_CFC_ (* Continuous Function Chart, elements in execution order *)
(* 50с *)
#0 INT_TO_TIME(SCHU_P2_3_YA2_ZADER_RAS_DOST)
#1 MUL(#0, 1000)
#2 TON_YA2_Rassog1:TON(IN: YA2_DOST, PT: #1)
#3 ABS(SCHU_P2_3_YA2_RASSOG)
#4 GT(#3, SCHU_P2_3_YA2_UST_RASSOG)
#5 GT(SCHU_P2_3_YA2_RASSOG, SCHU_P2_3_YA2_UST_RASSOG)
#6 SEL(SCHU_P2_3_UST_RE_STOP, #4, #5)
#7 ABS(SCHU_P2_3_YA2_RASSOG_POL)
#8 GT(#7, SCHU_P2_3_YA2_UST_RASSOG)
#9 AND(TRUE, #8)
#10 YA2_REG_POL <= #9
#11 SEL(YA2_REG_POL, #6, #8)
#12 AND(NOT SCHU_P2_3_UST_RE_PUSK, #11)
#13 INT_TO_TIME(SCHU_P2_3_YA2_ZADER_RAS)
#14 MUL(#13, 1000)
#15 TON_YA2_Rassog:TON(IN: #12, PT: #14)
#16 OR(#15.Q, YA2_AO_OTKAZ)
#17 AND(#2.Q, SCHU_P2_3_SA4_DI3_A, #16)
#18 SR_YA2_Otk:SR(SET1: #17, RESET: SCHU_P2_3_SB)
#19 SCHU_P2_3_Z_YA2_OTKAZ <= #18.Q1
_END_CFC_
(* the same logic as Structured Text *)
(* 50с *)
TON_YA2_Rassog1(IN := YA2_DOST, PT := INT_TO_TIME(SCHU_P2_3_YA2_ZADER_RAS_DOST) * 1000);
_t14 := ABS(SCHU_P2_3_YA2_RASSOG_POL) > SCHU_P2_3_YA2_UST_RASSOG;
YA2_REG_POL := TRUE AND _t14;
TON_YA2_Rassog(IN := NOT SCHU_P2_3_UST_RE_PUSK AND SEL(YA2_REG_POL, SEL(SCHU_P2_3_UST_RE_STOP, ABS(SCHU_P2_3_YA2_RASSOG) > SCHU_P2_3_YA2_UST_RASSOG, SCHU_P2_3_YA2_RASSOG > SCHU_P2_3_YA2_UST_RASSOG), _t14), PT := INT_TO_TIME(SCHU_P2_3_YA2_ZADER_RAS) * 1000);
SR_YA2_Otk(SET1 := TON_YA2_Rassog1.Q AND SCHU_P2_3_SA4_DI3_A AND (TON_YA2_Rassog.Q OR YA2_AO_OTKAZ), RESET := SCHU_P2_3_SB);
SCHU_P2_3_Z_YA2_OTKAZ := SR_YA2_Otk.Q1;
END_PROGRAM

(* POU TZBiS/TZB/Z_YA3_Otk, CFC *)
PROGRAM Z_YA3_Otk
VAR
	SR_YA3_Otk: SR;
	TON_YA3_Zakl: TON;
	TON_YA3_Rassog: TON;
END_VAR
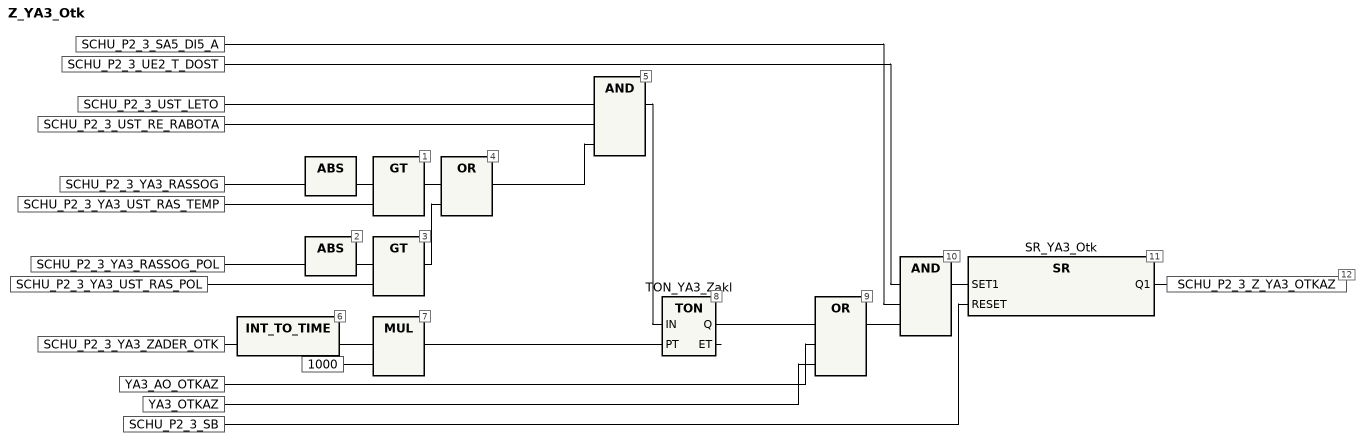
_CFC_ (* Continuous Function Chart, elements in execution order *)
#0 ABS(SCHU_P2_3_YA3_RASSOG)
#1 GT(#0, SCHU_P2_3_YA3_UST_RAS_TEMP)
#2 ABS(SCHU_P2_3_YA3_RASSOG_POL)
#3 GT(#2, SCHU_P2_3_YA3_UST_RAS_POL)
#4 OR(#1, #3)
#5 AND(SCHU_P2_3_UST_LETO, SCHU_P2_3_UST_RE_RABOTA, #4)
#6 INT_TO_TIME(SCHU_P2_3_YA3_ZADER_OTK)
#7 MUL(#6, 1000)
#8 TON_YA3_Zakl:TON(IN: #5, PT: #7)
#9 OR(#8.Q, YA3_AO_OTKAZ, YA3_OTKAZ)
#10 AND(SCHU_P2_3_UE2_T_DOST, SCHU_P2_3_SA5_DI5_A, #9)
#11 SR_YA3_Otk:SR(SET1: #10, RESET: SCHU_P2_3_SB)
#12 SCHU_P2_3_Z_YA3_OTKAZ <= #11.Q1
_END_CFC_
(* the same logic as Structured Text *)
TON_YA3_Zakl(IN := SCHU_P2_3_UST_LETO AND SCHU_P2_3_UST_RE_RABOTA AND ((ABS(SCHU_P2_3_YA3_RASSOG) > SCHU_P2_3_YA3_UST_RAS_TEMP) OR (ABS(SCHU_P2_3_YA3_RASSOG_POL) > SCHU_P2_3_YA3_UST_RAS_POL)), PT := INT_TO_TIME(SCHU_P2_3_YA3_ZADER_OTK) * 1000);
SR_YA3_Otk(SET1 := SCHU_P2_3_UE2_T_DOST AND SCHU_P2_3_SA5_DI5_A AND (TON_YA3_Zakl.Q OR YA3_AO_OTKAZ OR YA3_OTKAZ), RESET := SCHU_P2_3_SB);
SCHU_P2_3_Z_YA3_OTKAZ := SR_YA3_Otk.Q1;
END_PROGRAM

(* POU TZBiS/TZB/Z_YA4_Otk, CFC *)
PROGRAM Z_YA4_Otk
VAR
	RS_YA4_OTKZ: SR;

	UE3_ZADER: TON;
	SCHU_P2_3_YA4_AO4ER: TON;
	F_trig_ai: F_TRIG;
	TON_YA4: TON;
	YA4_ZADER_POL: TON;
	YA4_ZADER_TEMP: TON;
END_VAR
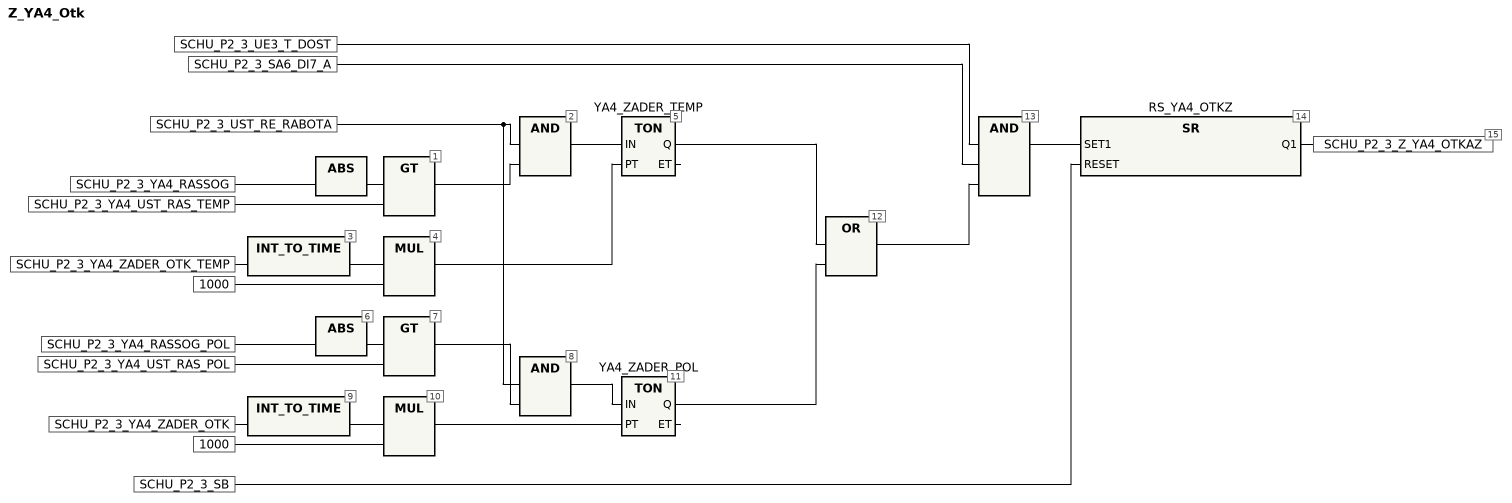
